// TIA Portal project "first_prj" (V17)

(* hardware
DEVICE "S7-1500/ET200MP station_1"  S7-1500 station
   slot 0: "Rail_0"  Rack  6ES7 590-1***0-0AA0
   slot 0: "PM 70W 120/230VAC"  PM 70W 120/230VAC  6EP1332-4BA00
   slot 1: "PLC_1"  CPU 1513F-1 PN  6ES7 513-1FL01-0AB0  V2.1
      slot 3: "CPU display_1"  6ES7591-1AA00-0AA0
      slot 32768: "PROFINET interface_1"  X1
         slot 32769: "Port_1"  X1 P1
         slot 32770: "Port_2"  X1 P2
   slot 2: "DI 32x24VDC HF_1"  DI 32x24VDC HF  6ES7 521-1BL00-0AB0  V2.1
   slot 3: "DQ 32x24VDC/0.5A HF_1"  DQ 32x24VDC/0.5A HF  6ES7 522-1BL01-0AB0  V1.0
   slot 4: "AI 8xU/I/RTD/TC ST_1"  AI 8xU/I/RTD/TC ST  6ES7 531-7KF00-0AB0  V2.0
DEVICE "ET 200SP station_1"  ET 200SP-Station
   slot 0: "Rack_0"  Rack  6ES5 710-8MAx1
   slot 0: "IO device_1"  IM 155-6 PN ST  6ES7 155-6AU00-0BN0  V3.3
   slot 1: "DI 8x24VDC ST_1"  DI 8x24VDC ST  6ES7 131-6BF00-0BA0  V1.1
      slot 1: "DI 8x24VDC ST_1"  DI 8x24VDC ST
   slot 2: "DI 8x24VDC ST_2"  DI 8x24VDC ST  6ES7 131-6BF00-0BA0  V1.1
      slot 1: "DI 8x24VDC ST_2"  DI 8x24VDC ST
   slot 3: "DQ 16x24VDC/0.5A ST_1"  DQ 16x24VDC/0.5A ST  6ES7 132-6BH00-0BA0  V1.1
      slot 1: "DQ 16x24VDC/0.5A ST_1"  DQ 16x24VDC/0.5A ST
   slot 4: "AI 4xU/I 2-wire ST_1"  AI 4xU/I 2-wire ST  6ES7 134-6HD00-0BA1  V1.1
      slot 1: "AI 4xU/I 2-wire ST_1"  AI 4xU/I 2-wire ST
   slot 5: "AQ 4xU/I ST_1"  AQ 4xU/I ST  6ES7 135-6HD00-0BA1  V1.1
      slot 1: "AQ 4xU/I ST_1"  AQ 4xU/I ST
   slot 6: "Server module_1"  Server module  6ES7 193-6PA00-0AA0  V1.1
      slot 1: "Server module_1"  Server module
   slot 127: "BA 2xRJ45"  BA 2xRJ45  6ES7 193-6AR00-0AA0  V0.0
      slot 1: "Port_1"  X1 P1 R  6ES7 193-6AR00-0AA0  V0.0
      slot 2: "Port_2"  X1 P2 R  6ES7 193-6AR00-0AA0  V0.0
DEVICE "HMI_1"  TP700 Comfort
   slot 0: "HMI_1"  TP700 Comfort  6AV2 124-0GC01-0AX0  17.0.0.0
   slot 1: "HMI_RT_1"  TP700 Comfort  6AV2 124-0GC01-0AX0  17.0.0.0
   slot 5: "HMI_1.IE_CP_1"  PROFINET Interface  17.0.0.0
      slot 1: "PROFINET Interface_1"  PROFINET Interface
         slot 1: "Port_1"  Port
         slot 2: "Port_2"  Port
   slot 7: "HMI_1.MPI/DP_CP_1"  MPI/DP Interface  17.0.0.0
*)

// ===== PLC "PLC_1"  CPU 1513F-1 PN =====

VAR_GLOBAL   // PLC tag table "Default tag table"
   "marker deny" AT %M0.0 : Bool;
   "btn1right" AT %M0.1 : Bool;
   "btn2right" AT %M0.2 : Bool;
   "switchs" AT %M0.3 : Bool;
   "go_right" AT %M0.4 : Bool;
   "auto_right" AT %M0.5 : Bool;
   "rising_con" AT %M0.6 : Bool;
   "rising 1" AT %M0.7 : Bool;
   "rising 2" AT %M1.0 : Bool;
   "all_markers" AT %M1.1 : Bool;
   "f1" AT %M10.5 : Bool;
   "f2" AT %M10.3 : Bool;
   "Tag_3" AT %M1.3 : Bool;
   "ack" AT %M3.0 : Bool;
   "out" AT %M4.0 : Bool;
   "F" AT %M4.1 : Bool;
   "A" AT %M4.2 : Bool;
   "condition_true" AT %M5.0 : Bool;
   "Tag_1" AT %M1.4 : Bool;
END_VAR

VAR_GLOBAL   // PLC tag table "Conveyor"
   "B_LB" AT %I4.0 : Bool;   // Lichtschranke / Light barrier
   "S_Bay1" AT %I4.1 : Bool;   // Taster Platz 1 / Momentary contact Bay 1
   "S_Bay2" AT %I4.2 : Bool;   // Taster Platz 2 / Momentary contact Bay 2
   "S_Bay3" AT %I4.3 : Bool;   // Taster Platz 3 / Momentary contact Bay 3
   "S_BayLB" AT %I4.4 : Bool;   // Taster Lichtschranken-Platz / Momentary contact Light barrier bay
   "B_Bay1" AT %I4.5 : Bool;   // Initiator Platz 1 / Proximity sensor Bay 1
   "B_Bay2" AT %I4.6 : Bool;   // Initiator Platz 2 / Proximity sensor Bay 2
   "B_Bay3" AT %I4.7 : Bool;   // Initiator Platz 3 / Proximity sensor Bay 3
   "P_Bay1" AT %Q4.1 : Bool;   // Meldeleuchte Platz 1 / Indicator light Bay 1
   "P_Bay2" AT %Q4.2 : Bool;   // Meldeleuchte Platz 2 / Indicator light Bay 2
   "P_Bay3" AT %Q4.3 : Bool;   // Meldeleuchte Platz 3 / Indicator light Bay 3
   "P_BayLB" AT %Q4.4 : Bool;   // Meldeleuchte Lichtschranken-Platz / Indicator light Light barrier bay
   "K_Right" AT %Q4.5 : Bool;   // Bandmotor Rechts / Run conveyor RIGHT
   "K_Left" AT %Q4.6 : Bool;   // Bandmotor Links / Run conveyor LEFT
   "P_Horn" AT %Q4.7 : Bool;   // Hupe / Horn
END_VAR

VAR_GLOBAL   // PLC tag table "My_Tags"
   "M_AuxLB" AT %M16.0 : Bool;   // Edge auxiliary memory bit Light barrier / Flanken-Hilfsmerker Lichtschranke
   "S_Fault3" AT %E0.6 : Bool;   // Schalter Störung 3 / S_Fault3
   "M_JogRight" AT %M16.2 : Bool;   // Merker Tippen Rechts / Memory bit Jog conveyor RIGHT
   "M_AutoRight" AT %M16.4 : Bool;   // Merker Auto Rechts / Memory bit Conveyor AUTO RIGHT
   "M_ConvFault" AT %M17.0 : Bool;   // Merker Bandlauf-Störung / Memory bit Conveyor fault
   "S_Acknowledge" AT %E0.7 : Bool;   // Taster Quittierung / S_Acknowledge
   "P_Operation" AT %A0.1 : Bool;   // Meldeleuchte Betrieb EIN / Indicator light Operation ON
   "P_Fault" AT %A0.7 : Bool;   // Anzeige Band-Störung / Indicator light for fault
   "M_AuxFault1" AT %M17.1 : Bool;   // Edge auxiliary memory bit Fault 1 / Flanken-Hilfsmerker Störung 1
   "P_Fault1" AT %A0.2 : Bool;   // Anzeige Störung 1 / Indicator light for fault1
   "P_Fault2" AT %A0.3 : Bool;   // Anzeige Störung 2 / Indicator light for fault2
   "S_Fault1" AT %E0.4 : Bool;   // Schalter Störung 1 / S_Fault1
   "S_Fault2" AT %E0.5 : Bool;   // Schalter Störung 2 / S_Fault2
   "P_Fault3" AT %A0.4 : Bool;   // Anzeige Störung 3 / Indicator light for fault3
   "M_AuxOpON" AT %M15.1 : Bool;   // Edge auxiliary memory bit Operation ON / Flanken-Hilfsmerker Anlage EIN
   "M_ActSetp" AT %M18.4 : Bool;   // Merker Ist-Stückzahl=Soll-Stückzah / Memory bit Actual- has reached Setpoint number
   "S_OperationON" AT %E0.1 : Bool;   // Taster Betrieb EIN / S_OperationON
   "S_OperationOFF" AT %E0.0 : Bool;   // Taster Betrieb AUS / S_OperationOFF
   "S_Right" AT %E0.2 : Bool;   // Taster Tippen Rechts / S_Right
   "S_Left" AT %E0.3 : Bool;   // Taster Tippen Links / S_Left
   "M_StorFault1" AT %M17.2 : Bool;   // Memory bit for storing Fault 1 / Merker Meldespeicher Störung 1
   "M_AuxFault2" AT %M17.3 : Bool;   // Edge auxiliary memory bit Fault 2 / Flanken-Hilfsmerker Störung 2
   "M_StorFault2" AT %M17.4 : Bool;   // Memory bit for storing Fault 2 / Merker Meldespeicher Störung 2
   "TOF-Timer-L" AT %M20.2 : Bool;
   "TOF-Timer-R" AT %M20.1 : Bool;
   "max_ConvFault" AT %M20.0 : Bool;
   "P_InitLeft" AT %A0.5 : Bool;
   "P_InitRight" AT %A0.6 : Bool;
   "S_Slider1" AT %IW10 : Word;
   "S_Slider2" AT %IW30 : Word;
END_VAR

VAR_GLOBAL CONSTANT   // PLC tag table "My_Tags"
   "const_maxTime" : Time := t#6s;   // max. Transportzeit / max. transport time
   "const_Setp" : UInt := 3;   // Sollwert / setpoint parts
END_VAR

DATA_BLOCK "HMI_Tags"   // DB1
{ S7_Optimized_Access := 'TRUE' }
VERSION : 0.1
   VAR
      Left_M : Bool;
      Right_M : Bool;
      S_BayLB : Bool;
      S_Bay3 : Bool;
      S_Bay2 : Bool;
      S_Bay1 : Bool;
   END_VAR
BEGIN
END_DATA_BLOCK

DATA_BLOCK "multiple_freq_mem_DB"   // DB2
{ S7_Optimized_Access := 'TRUE' }
VERSION : 0.1
// stored: InstanceOfName multiple_freq_mem
"multiple_freq_mem"
BEGIN
END_DATA_BLOCK

DATA_BLOCK "mfm2"   // DB3
{ S7_Optimized_Access := 'TRUE' }
VERSION : 0.1
BEGIN
END_DATA_BLOCK

DATA_BLOCK "parts_count_DB_2"   // DB4
{ S7_Optimized_Access := 'TRUE' }
VERSION : 0.1
// stored: InstanceOfName parts_count
"parts_count"
BEGIN
END_DATA_BLOCK

DATA_BLOCK "parts_count_DB"   // DB5
{ S7_Optimized_Access := 'TRUE' }
VERSION : 0.1
// stored: InstanceOfName parts_count
"parts_count"
BEGIN
END_DATA_BLOCK

DATA_BLOCK "parts_count_DB_1"   // DB6
{ S7_Optimized_Access := 'TRUE' }
VERSION : 0.1
// stored: InstanceOfName parts_count
"parts_count"
BEGIN
END_DATA_BLOCK

DATA_BLOCK "Data_block_1"   // DB7
{ S7_Optimized_Access := 'TRUE' }
VERSION : 0.1
BEGIN
END_DATA_BLOCK

DATA_BLOCK "data block 3"   // DB9
{ S7_Optimized_Access := 'TRUE' }
VERSION : 0.1
   VAR
      count : Int;
      fault : Bool;
      led : Bool;
      operation_off : Bool;
      operation_on : Bool;
      jog_right : Bool;
      jog_left : Bool;
      ack_fault : Bool;
      act_no : UInt;
      setp_no : UInt := 6;
   END_VAR
BEGIN
END_DATA_BLOCK

DATA_BLOCK "Data_block_2"   // DB10
{ S7_Optimized_Access := 'TRUE' }
VERSION : 0.1
BEGIN
END_DATA_BLOCK

// folder: System blocks/Program resources

DATA_BLOCK "IEC_Timer_0_DB_1"   // DB8
{ S7_Optimized_Access := 'TRUE' }
AUTHOR : Simatic
FAMILY : IEC
NAME : IEC_TMR
VERSION : 1.0
// stored: InstanceOfName IEC_TIMER
"IEC_TIMER"
BEGIN
END_DATA_BLOCK

// folder: (top level)

FUNCTION_BLOCK "multiple_freq_mem"   // FB1, LAD
{ S7_Optimized_Access := 'TRUE' }
VERSION : 0.1
   VAR_INPUT
      Fault : Bool;
      Acknowledge : Bool;
   END_VAR
   VAR_OUTPUT
      display : Bool;
   END_VAR
   VAR_IN_OUT
      Freq : Bool;
   END_VAR
   VAR
      mem : Bool;
   END_VAR
   VAR_TEMP   // added for the SCL form of the ladder/FBD networks
      _w1 : Bool;
   END_VAR
BEGIN

REGION Network 1
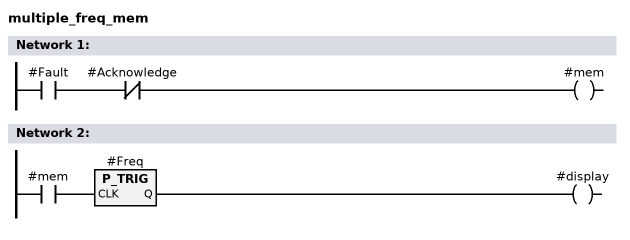
   RUNG wire#powerrail
      Contact( #Fault )
      I_Contact( #Acknowledge )
      Coil( #mem )
   END_RUNG
   // the same network as SCL:
   #mem := #Fault AND NOT #Acknowledge;
END_REGION

REGION Network 2
   RUNG wire#powerrail
      Contact( #mem )
      P_Trig( #Freq )
      Coil( #display )
   END_RUNG
   // the same network as SCL:
   #_w1 := #mem AND NOT #Freq;   // rising edge
   #Freq := #mem;
   #display := #_w1;
END_REGION
END_FUNCTION_BLOCK

FUNCTION_BLOCK "parts_count"   // FB2, LAD
{ S7_Optimized_Access := 'TRUE' }
VERSION : 0.1
   VAR_INPUT
      new_value : Int;
      max : Int := 5;
      sensor : Bool;
   END_VAR
   VAR_OUTPUT
      "Counter" : Int;
   END_VAR
   VAR
      Value : Int;
      Flag : Bool;
   END_VAR
   VAR RETAIN
      IEC_Counter_0_Instance : CTU_INT;
   END_VAR
   VAR_TEMP   // added for the SCL form of the ladder/FBD networks
      _w1 : Bool;
   END_VAR
BEGIN

REGION Network 1: S_Fault1
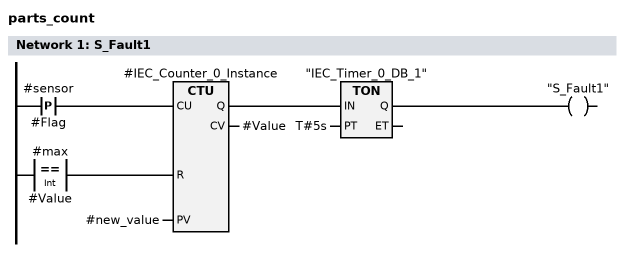
   #_w1 := #sensor AND NOT #Flag;   // rising edge of #sensor
   #Flag := #sensor;
   #IEC_Counter_0_Instance(CU := #_w1, R := #max = #Value, PV := #new_value, CV => #Value);   // CTU
   "IEC_Timer_0_DB_1".TON(IN := #IEC_Counter_0_Instance.Q, PT := T#5s);
   "S_Fault1" := "IEC_Timer_0_DB_1".Q;
END_REGION
END_FUNCTION_BLOCK

FUNCTION "CONVEYOR" : Void   // FC1, LAD
{ S7_Optimized_Access := 'TRUE' }
VERSION : 0.1
   VAR_TEMP   // added for the SCL form of the ladder/FBD networks
      _w1 : Bool;
   END_VAR
BEGIN

REGION Network 1: Run conveyor RIGHT
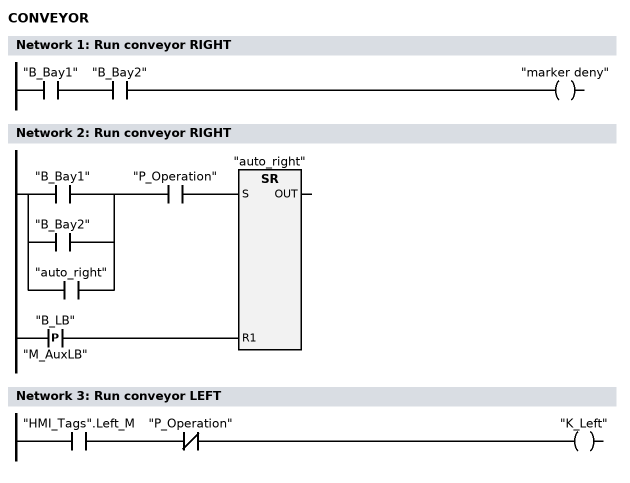
   RUNG wire#powerrail
      Contact( "B_Bay1" )
      Contact( "B_Bay2" )
      Coil( "marker deny" )
   END_RUNG
   // the same network as SCL:
   "marker deny" := "B_Bay1" AND "B_Bay2";
END_REGION

REGION Network 2: Run conveyor RIGHT
   RUNG wire#powerrail
      Contact( "B_Bay1" )
      wire#w1
      Contact( "P_Operation" )
      S_SR(operand := "auto_right", r1 := wire#w2)
   END_RUNG
   RUNG wire#powerrail
      Contact( "B_Bay2" )
   END_RUNG wire#w1
   RUNG wire#powerrail
      Contact( "auto_right" )
   END_RUNG wire#w1
   RUNG wire#powerrail
      P_Contact(operand := "B_LB", bit := "M_AuxLB")
   END_RUNG wire#w2
   // the same network as SCL:
   #_w1 := "B_LB" AND NOT "M_AuxLB";   // rising edge of "B_LB"
   "M_AuxLB" := "B_LB";
   IF ("B_Bay1" OR "B_Bay2" OR "auto_right") AND "P_Operation" THEN
       "auto_right" := TRUE;   // SR flip-flop
   END_IF;
   IF #_w1 THEN "auto_right" := FALSE; END_IF;
END_REGION

REGION Network 3: Run conveyor LEFT
   RUNG wire#powerrail
      Contact( "HMI_Tags".Left_M )
      I_Contact( "P_Operation" )
      Coil( "K_Left" )
   END_RUNG
   // the same network as SCL:
   "K_Left" := "HMI_Tags".Left_M AND NOT "P_Operation";
END_REGION
END_FUNCTION

FUNCTION "Fault_Det" : Void   // FC2, LAD
{ S7_Optimized_Access := 'TRUE' }
VERSION : 0.1
   VAR_INPUT
      P_Fault : Bool;
      S_Acknowledge : Bool;
   END_VAR
   VAR_OUTPUT
      Display : Bool;
   END_VAR
   VAR_IN_OUT
      Frequency : Bool;
   END_VAR
   VAR_TEMP
      ack : Bool;
      temp_mem : Bool;
      temp_2 : Bool;
   END_VAR
   VAR_TEMP   // added for the SCL form of the ladder/FBD networks
      _w1 : Bool;
   END_VAR
BEGIN

REGION Network 1
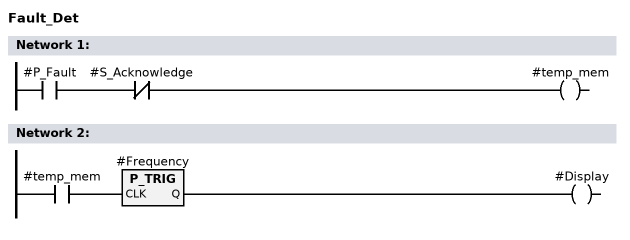
   RUNG wire#powerrail
      Contact( #P_Fault )
      I_Contact( #S_Acknowledge )
      Coil( #temp_mem )
   END_RUNG
   // the same network as SCL:
   #temp_mem := #P_Fault AND NOT #S_Acknowledge;
END_REGION

REGION Network 2
   RUNG wire#powerrail
      Contact( #temp_mem )
      P_Trig( #Frequency )
      Coil( #Display )
   END_RUNG
   // the same network as SCL:
   #_w1 := #temp_mem AND NOT #Frequency;   // rising edge
   #Frequency := #temp_mem;
   #Display := #_w1;
END_REGION
END_FUNCTION

ORGANIZATION_BLOCK "Main"   // OB1, LAD, ProgramCycle
TITLE = "Main Program Sweep (Cycle)"
{ S7_Optimized_Access := 'TRUE' }
VERSION : 0.1
   VAR_INPUT
      Initial_Call : Bool;   // Initial call of this OB
      Remanence : Bool;   // =True, if remanent data are available
   END_VAR
   VAR_TEMP
      SetPoint : Int;
      CV : Int;
   END_VAR
   VAR_TEMP   // added for the SCL form of the ladder/FBD networks
      _w1 : Bool;
   END_VAR
BEGIN

REGION Network 1: Indicator light Operation ON
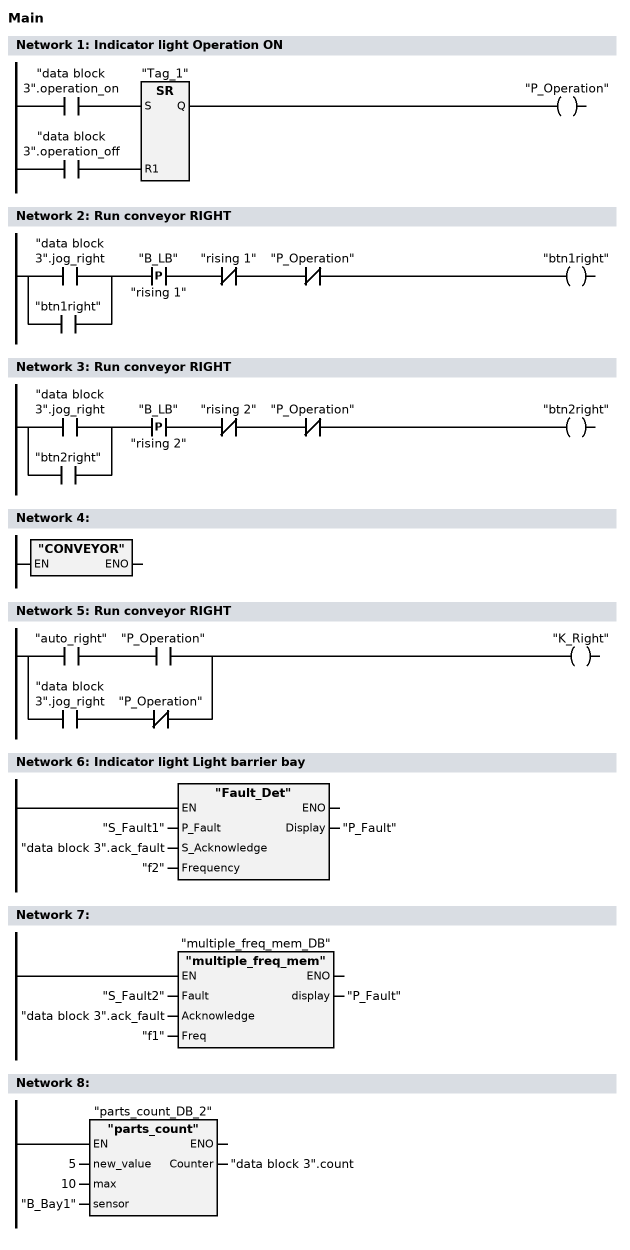
   RUNG wire#powerrail
      Contact( "data block 3".operation_on )
      S_SR(operand := "Tag_1", r1 := wire#w1)
      Coil( "P_Operation" )
   END_RUNG
   RUNG wire#powerrail
      Contact( "data block 3".operation_off )
   END_RUNG wire#w1
   // the same network as SCL:
   IF "data block 3".operation_on THEN
       "Tag_1" := TRUE;   // SR flip-flop
   END_IF;
   IF "data block 3".operation_off THEN "Tag_1" := FALSE; END_IF;
   "P_Operation" := "Tag_1";
END_REGION

REGION Network 2: Run conveyor RIGHT
   RUNG wire#powerrail
      Contact( "data block 3".jog_right )
      wire#w1
      P_Contact(operand := "B_LB", bit := "rising 1")
      I_Contact( "rising 1" )
      I_Contact( "P_Operation" )
      Coil( "btn1right" )
   END_RUNG
   RUNG wire#powerrail
      Contact( "btn1right" )
   END_RUNG wire#w1
   // the same network as SCL:
   #_w1 := ("data block 3".jog_right OR "btn1right") AND "B_LB" AND NOT "rising 1";   // rising edge of "B_LB"
   "rising 1" := "B_LB";
   "btn1right" := #_w1 AND NOT "rising 1" AND NOT "P_Operation";
END_REGION

REGION Network 3: Run conveyor RIGHT
   RUNG wire#powerrail
      Contact( "data block 3".jog_right )
      wire#w1
      P_Contact(operand := "B_LB", bit := "rising 2")
      I_Contact( "rising 2" )
      I_Contact( "P_Operation" )
      Coil( "btn2right" )
   END_RUNG
   RUNG wire#powerrail
      Contact( "btn2right" )
   END_RUNG wire#w1
   // the same network as SCL:
   #_w1 := ("data block 3".jog_right OR "btn2right") AND "B_LB" AND NOT "rising 2";   // rising edge of "B_LB"
   "rising 2" := "B_LB";
   "btn2right" := #_w1 AND NOT "rising 2" AND NOT "P_Operation";
END_REGION

REGION Network 4
   RUNG wire#powerrail
      "CONVEYOR"()
   END_RUNG
   // the same network as SCL:
   "CONVEYOR"();
END_REGION

REGION Network 5: Run conveyor RIGHT
   RUNG wire#powerrail
      Contact( "auto_right" )
      Contact( "P_Operation" )
      wire#w1
      Coil( "K_Right" )
   END_RUNG
   RUNG wire#powerrail
      Contact( "data block 3".jog_right )
      I_Contact( "P_Operation" )
   END_RUNG wire#w1
   // the same network as SCL:
   "K_Right" := ("auto_right" AND "P_Operation") OR ("data block 3".jog_right AND NOT "P_Operation");
END_REGION

REGION Network 6: Indicator light Light barrier bay
   RUNG wire#powerrail
      "Fault_Det"(P_Fault := "S_Fault1", S_Acknowledge := "data block 3".ack_fault, Frequency := "f2", Display => "P_Fault")
   END_RUNG
   // the same network as SCL:
   "Fault_Det"(P_Fault := "S_Fault1",
               S_Acknowledge := "data block 3".ack_fault,
               Frequency := "f2",
               Display => "P_Fault");
END_REGION

REGION Network 7
   RUNG wire#powerrail
      "multiple_freq_mem_DB"(Fault := "S_Fault2", Acknowledge := "data block 3".ack_fault, Freq := "f1", display => "P_Fault")
   END_RUNG
   // the same network as SCL:
   "multiple_freq_mem_DB"(Fault := "S_Fault2",   // "multiple_freq_mem"
                          Acknowledge := "data block 3".ack_fault,
                          Freq := "f1",
                          display => "P_Fault");
END_REGION

REGION Network 8
   RUNG wire#powerrail
      "parts_count_DB_2"(new_value := 5, max := 10, sensor := "B_Bay1", "Counter" => "data block 3".count)
   END_RUNG
   // the same network as SCL:
   "parts_count_DB_2"(new_value := 5, max := 10, sensor := "B_Bay1", "Counter" => "data block 3".count);   // "parts_count"
END_REGION
END_ORGANIZATION_BLOCK

(* ===== HMI "HMI_RT_1" =====
system functions are stored by id; their names below are inferred from use
connection "HMI_Connection_1": ETHERNET, S7_1500_OMS

HMI tags "Default tag table"
   "HMI_Plant_Off" : Bool = PLC "data block 3".operation_off AT %DB1.DBX0.0, 1 s
   "HMI_plant_On" : Bool = PLC "data block 3".operation_on AT %DB1.DBX0.0, 1 s
   "HMI_Jop_Right" : Bool = PLC "data block 3".jog_right AT %DB1.DBX0.0, 1 s
   "HMI_Jop_Left" : Bool = PLC "data block 3".jog_left AT %DB1.DBX0.0, 1 s
   "HMI_ACK_Fault" : Bool = PLC "data block 3".ack_fault AT %DB1.DBX0.0, 1 s
   "HMI_Set_Point" : UInt = PLC "data block 3".setp_no AT %DB1.DBX0.0, 1 s
   "HMI_Act_Number" : UInt = PLC "data block 3".act_no AT %DB1.DBX0.0, 1 s

Template "Template_1" 800x420
   Button "Alarms" at 720,2 size 78x58; TextOff 'Alarms'; PictureOff "AlarmDisplay_TP700_Comfort_TR"; PictureOn "AlarmDisplay_TP700_Comfort_TR"
      on Release: function_ef3f5d25("Alarm window_Unacknowledged", -1)
   Button "Template_Button" at 720,62 size 78x58; TextOff 'Text'
   Button "Template_Button_1" at 720,121 size 78x58; TextOff 'Text'
   Button "Template_Button_2" at 720,181 size 78x58; TextOff 'Text'
   Button "Template_Button_3" at 720,241 size 78x58; TextOff 'Text'
   Button "Template_Button_4" at 720,301 size 78x58; TextOff 'Text'
   Button "Template_Button_5" at 720,360 size 78x58; TextOff 'Text'

screen "Screen_1" 800x420
   Button "Button_1" at 64,63 size 96x32; TextOff 'Palnt On'
      on Press: SetBit("HMI_plant_On")
      on Release: ResetBit("HMI_plant_On")
   Button "Button_2" at 590,63 size 96x32; TextOff 'Plant Off'
      on Press: SetBit("HMI_Plant_Off")
      on Release: ResetBit("HMI_Plant_Off")
   Button "Button_3" at 61,186 size 96x32; TextOff 'Jop Right'
      on Press: SetBit("HMI_Jop_Right")
      on Release: ResetBit("HMI_Jop_Right")
   Button "Button_4" at 587,186 size 96x32; TextOff 'Jop Left'
      on Press: SetBit("HMI_Jop_Left")
      on Release: ResetBit("HMI_Jop_Left")
   Button "Button_5" at 62,342 size 96x32; TextOff 'Ack Fault'
      on Press: SetBit("HMI_ACK_Fault")
      on Release: ResetBit("HMI_ACK_Fault")
   IOField "I/O field_1" at 207,186 size 96x32; FormatPattern 99999
      ProcessValue <- "HMI_Set_Point"
   IOField "I/O field_2" at 443,186 size 96x32; FormatPattern 99999
      ProcessValue <- "HMI_Act_Number"
   TextField "Text field_1" at 202,154 size 89x23; Text 'Set Point'
   TextField "Text field_2" at 443,154 size 122x23; Text 'Actual Count'
*)